//==================================================================================================
//							Beckhoff Automation Poland
//									28.03.2018
//	Blok funkcyjny tworzacy strukture ST_DriveRef z AXIS_REF
//	Przydatny w komunikacji CoE w AX8000
//  v1.0	|| TC v 3.1.4022.16		|| - pierwsza wersja
//==================================================================================================
FUNCTION_BLOCK FB_GetDriveRef
VAR_INPUT
	bExecute								: BOOL;							// rising edge starts sequence
END_VAR
VAR_OUTPUT
	bBusy									: BOOL;
	bError									: BOOL;	
	udiErrorID								: UDINT;						// bError=TRUE AND udiErrorID=0 means state request timeout
	stDriveRef								: ST_DriveRef;					// come from stPlcDriveRef
END_VAR
VAR_IN_OUT
	Axis									: AXIS_REF;
END_VAR
VAR
	fbAdsRead								: ADSREAD;
	ftADSRead								: F_TRIG;
	stPlcDriveRef							: ST_PlcDriveRef;				// ADS buffer (need to change aNetId into sNetId)
END_VAR
VAR CONSTANT
	NCIDXG_AXPARMS							: UDINT			:= 16#4000;		// ADS group number to axis parameters 
	NCIDXO_AXP_HWAMSADDR					: UDINT			:= 16#31;		// ADS offset to drive channel
END_VAR

fbAdsRead(	NETID			:= '', 
			PORT			:= AMSPORT_R0_NC, 								// set ADS Port to NC
			IDXGRP			:= NCIDXG_AXPARMS + Axis.NcToPlc.AxisId,		// set ADS Group to AXIS Parameters 
			IDXOFFS			:= NCIDXO_AXP_HWAMSADDR,						// set ADS offset to channel number 
			LEN				:= SIZEOF(stPlcDriveRef), 
			DESTADDR		:= ADR(stPlcDriveRef), 
			READ			:= bExecute, 
			BUSY			=> bBusy, 
			ERR				=> bError, 
			ERRID			=> udiErrorID);
			
ftADSRead(CLK:= bBusy);

IF ftADSRead.Q AND NOT fbAdsRead.ERR THEN	
	stDriveRef.sNetId		:= F_CreateAmsNetId(stPlcDriveRef.aNetId);		// change AmsNetId array into string
	stDriveRef.nSlaveAddr	:= stPlcDriveRef.nSlaveAddr;
	stDriveRef.nDriveNo		:= stPlcDriveRef.nDriveNo;			
END_IF

END_FUNCTION_BLOCK

(* stored: Version 1.1.0.1, ProductVersion 3.1.4026.13, FileIdentifier 934b75291841a7adb6a18e0e3ac1cf3a29b894a2, FileSignature 18adc41fbe09ccc0be296cfe43abcac22e9c916f1c4ff3c5401811885d284f7e6bde1ec0985643f80bfe78bd0be780fb58ee3887f2490ed9ca858444b0a22903311a7ab4838363d740d239eca004fe91f2ff252f31a4a73bbbb51f152b5b3d691edc4f7654c84ed7ad63294f65301aad38a02012776c5b2c83ede96a13125ce7f741d444b1af4c983397f6c5ae13ef75ac64ea07de55eae8aa9489c4e96384e0cc3851c71d018596e682e85cb4cb7067e933e22516f72484554f0996f9c166fcbd0261582edf5a36b14882e44fbebb0dff0f66eaf73b695c5077738c559e5adb072e42b857d2bf83cf39df0dd7864a06ce5cb052e5be19d816369eb3c3f81ff2
   POU FB_GetDriveRef: Id {8789b1f0-f301-49cd-bbfe-fee0e4d04569}, SpecialFunc None *)
